{attribute 'qualified_only'}
VAR_GLOBAL
    HydraulicPumpRunningLamp  AT %Q* : BOOL;
END_VAR

(* stored: Version 1.1.0.1, ProductVersion 3.1.4024.9
   GVL DigitalOutputs: Id {00222bf0-a1a8-45d2-a046-556525ac83f5} *)
